Universal Robots PolyScope program: 0622_1902.urp

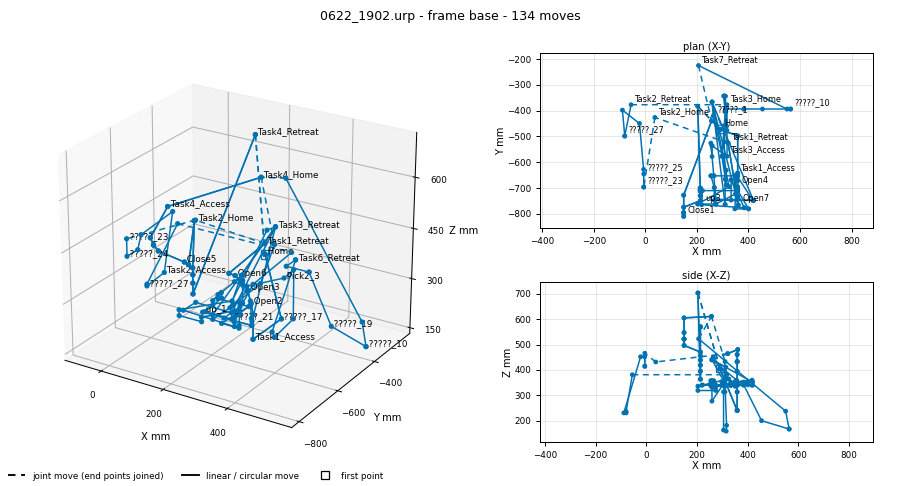
[picture p0: tool path of 0622_1902.urp in frame base, 134 of 134 moves have a stored position in this frame; points joined in program order, loops and branches not executed]
Program 0622_1902 (installation=default directory=/programs/usbdisk/새로운 폴더_3 createdIn=5.12.7.1102192 lastSavedIn=5.11.0.108249 robotSerialNumber=20215501208)
Calibrated DH parameters: a=[0.000135, -0.201821, -0.391913, -0.000063, 0.000038, 0]; d=[0.162484, -479.507804, 481.562221, -1.92078, 0.099549, 0.099572]; alpha=[1.570789, -0.00078, 0.007148, 1.569147, -1.569841, 0]; deltaTheta=[0, 1.075971, -1.038513, -0.037456, 0, 0]
Robot Program (runOnlyOnce=false)
  Folder Init
    Call Init_Variables
    Script: global repeat = 0
    Call Socket_Open
    MoveJ speed 60 deg/s, acceleration 80 deg/s^2 (useActiveTCP=true) feature=Base
      Waypoint Home: TCP in base x=290.307 y=-472.673 z=405.346 mm, rx=-2.2604 ry=-2.147 rz=0.0783 rad; joints [-251.839, -82.418, 93.917, 258.527, -92.811, 111.318] deg
    Wait Sleep waitTime=1
  Loop Forever
    Folder Main Sequence
      Folder Task1:OpenPrinter
        Call Enter_Next_Task
        Loop While (checkContinuously=false) expression=retry_count <= max_retry and task_done == 0
          MoveJ speed 60 deg/s, acceleration 80 deg/s^2 (useActiveTCP=true) feature=Base
            Waypoint Task1_Home: TCP in base x=290.314 y=-472.7 z=405.337 mm, rx=-2.2604 ry=-2.147 rz=0.0783 rad; joints [-251.84, -82.414, 93.913, 258.528, -92.81, 111.316] deg
          MoveL speed 250 mm/s, acceleration 1200 mm/s^2 (useActiveTCP=true) feature=Base
            Waypoint 웨이포인트_17: TCP in base x=358.108 y=-497.437 z=239.959 mm, rx=-2.2605 ry=-2.1469 rz=0.0783 rad; joints [-246.378, -66.361, 98.95, 237.748, -92.865, 116.914] deg
            Waypoint Task1_Access: TCP in base x=358.145 y=-643.31 z=239.914 mm, rx=-2.2603 ry=-2.1469 rz=0.0783 rad; joints [-250.947, -51.356, 74.514, 246.926, -92.843, 112.267] deg
          MoveL speed 250 mm/s, acceleration 1200 mm/s^2 (useActiveTCP=true) feature=Base
            Waypoint Open1: TCP in base x=358.112 y=-643.249 z=312.941 mm, rx=-2.2756 ry=-2.1607 rz=0.0433 rad; joints [-251.165, -54.868, 69.274, 255.167, -91.168, 112.004] deg
            Waypoint Open2: TCP in base x=358.116 y=-653.358 z=348.764 mm, rx=-2.2399 ry=-2.1285 rz=-0.0282 rad; joints [-251.571, -53.878, 61.395, 265.654, -89.944, 111.495] deg
            Waypoint Open3: TCP in base x=358.131 y=-671.047 z=394.191 mm, rx=-2.2065 ry=-2.0982 rz=-0.0914 rad; joints [-252.118, -50.739, 48.753, 278.451, -88.91, 110.769] deg
            Waypoint Open4: TCP in base x=358.139 y=-695.842 z=432.417 mm, rx=-2.2066 ry=-2.0983 rz=-0.0912 rad; joints [-252.66, -45.306, 33.722, 288.051, -88.986, 110.159] deg
            Waypoint Open5: TCP in base x=358.138 y=-703.871 z=432.339 mm, rx=2.1752 ry=2.0611 rz=-0.2397 rad; joints [-252.159, -50.267, 46.998, 262.355, -94.486, 110.613] deg
            Waypoint Open6: TCP in base x=358.152 y=-732.149 z=460.497 mm, rx=2.1751 ry=2.0611 rz=-0.2398 rad; joints [-252.775, -44.157, 32.21, 270.972, -94.36, 109.938] deg
            Waypoint Open7: TCP in base x=360.469 y=-765.799 z=480.398 mm, rx=2.1073 ry=1.9941 rz=-0.3503 rad; joints [-253.083, -35.969, 16.049, 272.511, -96.174, 109.139] deg
          MoveL speed 250 mm/s, acceleration 1200 mm/s^2 (useActiveTCP=true) feature=Base
            Waypoint Task1_Retreat: TCP in base x=320.913 y=-525.366 z=464.12 mm, rx=-2.2348 ry=-2.2055 rz=-0.1004 rad; joints [-251.676, -74.86, 75.667, 270.873, -86.355, 109.144] deg
          Wait Sleep waitTime=1
          SuppressedNode
            Call Check_Door_Open
          SuppressedNode
            Switch expression=fail_flag
              Case (caseValue=0)
                Script: task_done = 1
              Case (caseValue=1)
                Script: retry_count = retry_count + 1
          Call Check_Camera_Open
          Switch expression=fail_flag
            Case (caseValue=0)
              Script: task_done = 1
            Case (caseValue=1)
              Script: retry_count = retry_count + 1
        If task_done == 0
          Call Error_Stop
        Wait Sleep waitTime=1
      Folder Task2,3,3+:PickAndPlace
        Call Enter_Next_Task
        Loop While (checkContinuously=false) expression=nopaper == 1
          Loop While (checkContinuously=false) expression=retry_count <= max_retry and task_done == 0
            Folder Task2:PickA4FromTray
              MoveJ speed 60 deg/s, acceleration 80 deg/s^2 (useActiveTCP=true) feature=Base
                Waypoint Task2_Home: TCP in base x=36.96 y=-426.094 z=431.249 mm, rx=1.9338 ry=1.8099 rz=-0.6845 rad; joints [-284.402, -104.722, 122.782, 215.162, -85.651, 81.217] deg
              Call Gripper_Open
              Call Wait_Motor_Idle
              Folder 폴더
                MoveJ speed 60 deg/s, acceleration 80 deg/s^2 (useActiveTCP=true) feature=Base
                  Waypoint 웨이포인트_23: TCP in base x=-6.335 y=-696.326 z=465.636 mm, rx=2.2415 ry=-0.3574 rz=-0.16 rad; joints [-280.885, -66.992, 81.728, 205.322, -95.11, 185.235] deg
                MoveL speed 250 mm/s, acceleration 1200 mm/s^2 (useActiveTCP=true) feature=Base
                  Waypoint 웨이포인트_24: TCP in base x=-6.322 y=-696.307 z=414.387 mm, rx=2.2415 ry=-0.3575 rz=-0.16 rad; joints [-280.889, -64.814, 86.427, 198.445, -95.156, 185.249] deg
                  Waypoint 웨이포인트_25: TCP in base x=-6.303 y=-645.419 z=414.389 mm, rx=2.2414 ry=-0.3575 rz=-0.16 rad; joints [-281.881, -71.275, 95.746, 195.526, -94.416, 184.618] deg
                  Waypoint 웨이포인트_28: TCP in base x=-6.918 y=-627.811 z=451.854 mm, rx=2.2414 ry=-0.3575 rz=-0.1599 rad; joints [-282.329, -75.473, 95.437, 200.006, -94.042, 184.326] deg
              MoveL speed 250 mm/s, acceleration 1200 mm/s^2 (useActiveTCP=true) feature=Base
                Waypoint 웨이포인트_26: TCP in base x=-22.834 y=-449.606 z=451.838 mm, rx=2.2414 ry=-0.3575 rz=-0.1599 rad; joints [-290.868, -100.504, 121.499, 198.842, -87.496, 178.874] deg
                Waypoint Task2_Access: TCP in base x=-89.035 y=-397.687 z=230.223 mm, rx=1.5681 ry=0.0538 rz=0.0669 rad; joints [-313.235, -57.01, 139.142, 97.671, -42.763, 180.679] deg
                Waypoint 웨이포인트_27: TCP in base x=-80.06 y=-498.27 z=230.219 mm, rx=1.5682 ry=0.0538 rz=0.067 rad; joints [-301.557, -52.728, 123.378, 109.146, -54.422, 180.732] deg
                Waypoint 웨이포인트_12: TCP in base x=-80.054 y=-498.26 z=235.695 mm, rx=1.5681 ry=0.0538 rz=0.0669 rad; joints [-301.558, -53.562, 123.445, 109.909, -54.42, 180.737] deg
              Wait Sleep waitTime=1
              Call Gripper_Close
              Call Wait_Motor_Idle
              MoveL speed 250 mm/s, acceleration 1200 mm/s^2 (useActiveTCP=true) feature=Base
                Waypoint Task2_Retreat: TCP in base x=-55.478 y=-376.727 z=380.943 mm, rx=1.5681 ry=0.0539 rz=0.0669 rad; joints [-310.988, -89.069, 140.295, 128.379, -44.954, 180.96] deg
              If fail_flag == 1
                Call Error_Stop
              Wait Sleep waitTime=3
            Folder Task3:PlaceA4OnScanner
              Call Enter_Next_Task
              MoveJ speed 60 deg/s, acceleration 80 deg/s^2 (useActiveTCP=true) feature=Base
                Waypoint Task3_Home: TCP in base x=316.751 y=-376.736 z=380.91 mm, rx=1.5682 ry=0.054 rz=0.0668 rad; joints [-240.78, -72.729, 119.686, 133.121, -115.13, 180.786] deg
              MoveL speed 250 mm/s, acceleration 1200 mm/s^2 (useActiveTCP=true) feature=Base
                Waypoint Task3_Access: TCP in base x=316.801 y=-576.799 z=363.883 mm, rx=1.5682 ry=0.054 rz=0.067 rad; joints [-250.736, -54.554, 93.02, 141.565, -105.113, 180.827] deg
              MoveL speed 250 mm/s, acceleration 1200 mm/s^2 (useActiveTCP=true) feature=Base
                Waypoint Place1: TCP in base x=258.695 y=-535.855 z=276.647 mm, rx=1.5682 ry=0.0539 rz=0.067 rad; joints [-255.555, -52.152, 107.026, 125.111, -100.371, 180.737] deg
                Waypoint Place2: TCP in base x=258.714 y=-535.837 z=330.851 mm, rx=1.9481 ry=0.0428 rz=0.0806 rad; joints [-255.789, -65.713, 110.061, 157.638, -98.984, 186.181] deg
                Waypoint Place3: TCP in base x=258.706 y=-577.686 z=357.608 mm, rx=2.0696 ry=0.0386 rz=0.0849 rad; joints [-257.026, -66.21, 102.611, 172.482, -97.075, 187.174] deg
              Call Gripper_Open
              Call Wait_Motor_Idle
              MoveL speed 250 mm/s, acceleration 1200 mm/s^2 (useActiveTCP=true) feature=Base
                Waypoint 웨이포인트_6: TCP in base x=254.047 y=-525.754 z=357.577 mm, rx=2.1241 ry=0.0396 rz=0.0817 rad; joints [-256.235, -72.651, 110.764, 173.964, -97.528, 187.976] deg
                Waypoint 웨이포인트_7: TCP in base x=265.506 y=-653.622 z=357.598 mm, rx=2.124 ry=0.0397 rz=0.0817 rad; joints [-258.032, -58.705, 89.296, 181.36, -95.938, 187.013] deg
                Waypoint 웨이포인트_8: TCP in base x=265.302 y=-651.492 z=340.681 mm, rx=2.124 ry=0.0397 rz=0.0817 rad; joints [-258.01, -57.739, 90.591, 179.098, -95.971, 187.023] deg
                Waypoint 웨이포인트_13: TCP in base x=273.53 y=-743.632 z=340.722 mm, rx=2.124 ry=0.0397 rz=0.0817 rad; joints [-258.911, -46.995, 71.73, 187.158, -95.142, 186.541] deg
                Waypoint 웨이포인트_21: TCP in base x=356.126 y=-746.074 z=340.698 mm, rx=2.124 ry=0.0397 rz=0.0818 rad; joints [-252.554, -42.043, 62.558, 191.888, -100.492, 189.948] deg
                Waypoint 웨이포인트_29: TCP in base x=356.13 y=-746.059 z=359.504 mm, rx=2.124 ry=0.0397 rz=0.0817 rad; joints [-252.552, -43.007, 61.421, 193.988, -100.482, 189.944] deg
              MoveL speed 250 mm/s, acceleration 1200 mm/s^2 (useActiveTCP=true) feature=Base
                Waypoint Task3_Retreat: TCP in base x=258.692 y=-366.204 z=439.923 mm, rx=2.1237 ry=0.0367 rz=0.0867 rad; joints [-249.2, -96.96, 123.493, 186.236, -103.267, 192.051] deg
              Wait Sleep waitTime=1
              Call Check_Camera_Align
              Switch expression=paper_state
                Case (caseValue=0)
                  Script: retry_count = retry_count + 1
                Case (caseValue=1)
                  Script: task_done = 1
              Wait Sleep waitTime=1
          If task_done == 0
            Call Error_Stop
          Folder Task3+:PaperAlign
            Wait Sleep waitTime=1
            Call Check_Camera_Align
            Loop While (checkContinuously=false) expression=paper_align_state != 0 and paper_align_state != 9 and align_retry_count <= max_retry
              Script: align_retry_count = align_retry_count + 1
              MoveL speed 250 mm/s, acceleration 1200 mm/s^2 (useActiveTCP=true) feature=Base
                Waypoint 웨이포인트_1: TCP in base x=263.645 y=-419.544 z=450.752 mm, rx=2.1095 ry=0.0567 rz=0.0671 rad; joints [-251.124, -90.818, 116.42, 186.206, -102.101, 189.536] deg
                Waypoint 웨이포인트_5: TCP in base x=325.163 y=-694.866 z=364.547 mm, rx=2.1237 ry=0.0368 rz=0.0868 rad; joints [-253.782, -51.437, 75.758, 187.916, -99.351, 189.514] deg
              Switch expression=paper_align_state
                Case (caseValue=1)
                  SuppressedNode
                    MoveL speed 250 mm/s, acceleration 1200 mm/s^2 (useActiveTCP=true) feature=Base
                      Waypoint home_up: TCP in base x=411.069 y=-776.712 z=349.862 mm, rx=2.1238 ry=0.0368 rz=0.0867 rad; joints [-249.41, -33.925, 45.774, 200.882, -102.945, 191.884] deg
                      Waypoint touch: TCP in base x=411.033 y=-776.714 z=334.504 mm, rx=2.1236 ry=0.0367 rz=0.0867 rad; joints [-249.413, -33.291, 46.859, 199.158, -102.957, 191.886] deg
                      Waypoint down: TCP in base x=313.835 y=-617.619 z=339.178 mm, rx=2.1238 ry=0.0367 rz=0.0868 rad; joints [-252.767, -58.652, 92.334, 178.663, -100.285, 190.075] deg
                      Waypoint right: TCP in base x=250.722 y=-620.02 z=338.484 mm, rx=2.1239 ry=0.0366 rz=0.0869 rad; joints [-258.809, -61.528, 97.303, 176.099, -95.176, 186.838] deg
                      Waypoint up: TCP in base x=245.21 y=-744.892 z=339.67 mm, rx=2.1238 ry=0.0367 rz=0.0868 rad; joints [-261.255, -48.066, 73.863, 185.967, -93.018, 185.539] deg
                      Waypoint left: TCP in base x=408.353 y=-753.62 z=337.643 mm, rx=2.1235 ry=0.0364 rz=0.0868 rad; joints [-248.997, -37.091, 53.665, 196.203, -103.338, 192.136] deg
                      Waypoint z_up: TCP in base x=408.373 y=-753.612 z=350.303 mm, rx=2.1236 ry=0.0365 rz=0.0868 rad; joints [-248.995, -37.678, 52.851, 197.607, -103.325, 192.135] deg
                  SuppressedNode
                    MoveL speed 250 mm/s, acceleration 1200 mm/s^2 (useActiveTCP=true) feature=Base
                      Waypoint top_home: TCP in base x=476.403 y=-777.08 z=332.173 mm, rx=2.0259 ry=0.0603 rz=0.0427 rad; joints [-244.874, -24.378, 31.553, 200.812, -109.067, 190.542] deg
                      Waypoint lefttop1: TCP in base x=476.428 y=-777.056 z=326.289 mm, rx=2.0258 ry=0.0603 rz=0.0427 rad; joints [-244.872, -24.18, 32.025, 200.14, -109.072, 190.543] deg
                      Waypoint lefttop2: TCP in base x=418.211 y=-735.241 z=318.888 mm, rx=2.0259 ry=0.0603 rz=0.0427 rad; joints [-247.527, -36.33, 57.095, 186.808, -106.819, 189.265] deg
                      Waypoint lefttop3: TCP in base x=418.224 y=-735.252 z=329.315 mm, rx=2.0259 ry=0.0603 rz=0.0428 rad; joints [-247.527, -36.912, 56.59, 187.895, -106.81, 189.264] deg
                      Waypoint lefttop4: TCP in base x=476.403 y=-777.08 z=332.173 mm, rx=2.0259 ry=0.0603 rz=0.0427 rad; joints [-244.874, -24.378, 31.553, 200.812, -109.067, 190.542] deg
                      Waypoint lefttop5: TCP in base x=476.428 y=-777.056 z=326.289 mm, rx=2.0258 ry=0.0603 rz=0.0427 rad; joints [-244.872, -24.18, 32.025, 200.14, -109.072, 190.543] deg
                      Waypoint lefttop6: TCP in base x=418.249 y=-735.21 z=317.328 mm, rx=2.0257 ry=0.0603 rz=0.0428 rad; joints [-247.524, -36.239, 57.167, 186.634, -106.822, 189.262] deg
                      Waypoint 웨이포인트_34: TCP in base x=254.455 y=-652.624 z=348.54 mm, rx=2.1239 ry=0.0371 rz=0.0867 rad; joints [-259.06, -58.691, 90.844, 179.708, -94.929, 186.683] deg
                      Waypoint move_to_right: TCP in base x=316.854 y=-733.109 z=330.021 mm, rx=2.0257 ry=-0.0559 rz=-0.0297 rad; joints [-254.229, -43.603, 69.178, 181.965, -106.74, 189.197] deg
                      Waypoint righttop_home: TCP in base x=198.901 y=-787.594 z=329.962 mm, rx=2.018 ry=-0.2066 rz=-0.1238 rad; joints [-263.364, -41.811, 65.831, 183.44, -106.194, 188.908] deg
                      Waypoint righttop1: TCP in base x=198.92 y=-787.585 z=321.803 mm, rx=2.018 ry=-0.2066 rz=-0.1238 rad; joints [-263.362, -41.311, 66.196, 182.574, -106.201, 188.907] deg
                      Waypoint righttop2: TCP in base x=198.916 y=-755.326 z=321.817 mm, rx=2.0181 ry=-0.2066 rz=-0.1237 rad; joints [-263.056, -45.33, 73.758, 179.077, -106.5, 189.056] deg
                      Waypoint 웨이포인트_35: TCP in base x=267.387 y=-698.175 z=352.437 mm, rx=2.1237 ry=0.0371 rz=0.0866 rad; joints [-258.698, -53.341, 81.09, 184.124, -95.208, 186.872] deg
                      Waypoint righttop_home: TCP in base x=198.901 y=-787.594 z=329.962 mm, rx=2.018 ry=-0.2066 rz=-0.1238 rad; joints [-263.364, -41.811, 65.831, 183.44, -106.194, 188.908] deg
                      Waypoint righttop1: TCP in base x=198.92 y=-787.585 z=321.803 mm, rx=2.018 ry=-0.2066 rz=-0.1238 rad; joints [-263.362, -41.311, 66.196, 182.574, -106.201, 188.907] deg
                      Waypoint righttop2: TCP in base x=198.916 y=-755.326 z=321.817 mm, rx=2.0181 ry=-0.2066 rz=-0.1237 rad; joints [-263.056, -45.33, 73.758, 179.077, -106.5, 189.056] deg
                      Waypoint 웨이포인트_35: TCP in base x=267.387 y=-698.175 z=352.437 mm, rx=2.1237 ry=0.0371 rz=0.0866 rad; joints [-258.698, -53.341, 81.09, 184.124, -95.208, 186.872] deg
                      Waypoint 웨이포인트_36: TCP in base x=267.318 y=-698.171 z=339.177 mm, rx=2.1237 ry=0.0369 rz=0.0866 rad; joints [-258.704, -52.477, 81.792, 182.558, -95.216, 186.875] deg
                      Waypoint 웨이포인트_37: TCP in base x=378.814 y=-710.052 z=321.31 mm, rx=2.0182 ry=-0.2066 rz=-0.1238 rad; joints [-247.983, -41.401, 65.997, 186.167, -119.675, 197.015] deg
                      Waypoint 웨이포인트_38: TCP in base x=378.85 y=-764.571 z=321.307 mm, rx=2.0182 ry=-0.2066 rz=-0.1238 rad; joints [-249.486, -34.393, 52.607, 192.111, -118.328, 196.135] deg
                      Waypoint 웨이포인트_39: TCP in base x=378.79 y=-764.605 z=321.308 mm, rx=2.0182 ry=-0.2067 rz=-0.1239 rad; joints [-249.491, -34.393, 52.605, 192.113, -118.329, 196.133] deg
                  MoveL speed 250 mm/s, acceleration 1200 mm/s^2 (useActiveTCP=true) feature=Base
                    Waypoint out_top_home_1: TCP in base x=203.102 y=-761.983 z=335.486 mm, rx=2.0028 ry=-0.2108 rz=-0.1158 rad; joints [-262.793, -45.047, 71.304, 180.396, -106.628, 189.392] deg
                    Waypoint out_top_touch_1: TCP in base x=203.111 y=-761.964 z=318.614 mm, rx=2.0027 ry=-0.2108 rz=-0.1159 rad; joints [-262.792, -43.949, 72.027, 178.57, -106.643, 189.389] deg
                    Waypoint out_top_left_1: TCP in base x=273.333 y=-761.997 z=318.66 mm, rx=2.0026 ry=-0.2109 rz=-0.1159 rad; joints [-257.196, -40.917, 66.151, 182.335, -111.608, 192.092] deg
                    Waypoint out_top_z_up_1: TCP in base x=273.301 y=-762.006 z=331.73 mm, rx=2.0027 ry=-0.2109 rz=-0.1159 rad; joints [-257.198, -41.724, 65.578, 183.721, -111.597, 192.093] deg
                    Waypoint out_top_home_2: TCP in base x=350.147 y=-722.859 z=353.835 mm, rx=2.1236 ry=0.0368 rz=0.0867 rad; joints [-252.473, -46.032, 67.835, 190.561, -100.442, 190.217] deg
                    Waypoint out_top_touch_2: TCP in base x=350.162 y=-722.849 z=335.209 mm, rx=2.1236 ry=0.0368 rz=0.0868 rad; joints [-252.473, -44.979, 68.869, 188.473, -100.452, 190.221] deg
                    Waypoint down_1: TCP in base x=350.105 y=-652.862 z=337.787 mm, rx=2.1238 ry=0.0368 rz=0.0868 rad; joints [-250.62, -52.889, 82.637, 182.839, -102.064, 191.242] deg
                    Waypoint right_1: TCP in base x=254.42 y=-652.638 z=336.904 mm, rx=2.1238 ry=0.037 rz=0.0867 rad; joints [-259.063, -57.835, 91.436, 178.254, -94.94, 186.683] deg
                    Waypoint 웨이포인트_34: TCP in base x=254.455 y=-652.624 z=348.54 mm, rx=2.1239 ry=0.0371 rz=0.0867 rad; joints [-259.06, -58.691, 90.844, 179.708, -94.929, 186.683] deg
                    Waypoint 웨이포인트_35: TCP in base x=267.387 y=-698.175 z=352.437 mm, rx=2.1237 ry=0.0371 rz=0.0866 rad; joints [-258.698, -53.341, 81.09, 184.124, -95.208, 186.872] deg
                    Waypoint 웨이포인트_36: TCP in base x=267.318 y=-698.171 z=339.177 mm, rx=2.1237 ry=0.0369 rz=0.0866 rad; joints [-258.704, -52.477, 81.792, 182.558, -95.216, 186.875] deg
                    Waypoint up_1: TCP in base x=267.384 y=-747.516 z=339.193 mm, rx=2.1237 ry=0.037 rz=0.0867 rad; joints [-259.485, -46.723, 71.497, 187.057, -94.512, 186.455] deg
                    Waypoint left_1: TCP in base x=417.039 y=-747.555 z=339.153 mm, rx=2.1238 ry=0.0369 rz=0.0866 rad; joints [-248.23, -37.306, 53.822, 196.381, -103.973, 192.544] deg
                    Waypoint z_up_2: TCP in base x=417.042 y=-747.569 z=359.498 mm, rx=2.1237 ry=0.0369 rz=0.0866 rad; joints [-248.228, -38.218, 52.46, 198.653, -103.963, 192.541] deg
                Case (caseValue=2)
                  MoveL speed 250 mm/s, acceleration 1200 mm/s^2 (useActiveTCP=true) feature=Base
                    Waypoint out_down_home: motionParameters(nextMotionTime=2); TCP in base x=353.061 y=-649.128 z=353.349 mm, rx=2.1237 ry=0.0367 rz=0.0867 rad; joints [-250.263, -54.126, 82.18, 184.573, -102.361, 191.44] deg
                    Waypoint out_down_touch: TCP in base x=353.03 y=-649.115 z=339.829 mm, rx=2.1237 ry=0.0367 rz=0.0867 rad; joints [-250.265, -53.239, 82.9, 182.965, -102.368, 191.441] deg
                    Waypoint up2: TCP in base x=347.298 y=-780.895 z=340.744 mm, rx=2.1237 ry=0.0368 rz=0.0868 rad; joints [-253.981, -37.91, 54.824, 195.3, -99.119, 189.395] deg
                    Waypoint left2: TCP in base x=400.466 y=-780.911 z=340.74 mm, rx=2.1237 ry=0.0368 rz=0.0868 rad; joints [-250.239, -33.821, 46.958, 199.482, -102.253, 191.428] deg
                    Waypoint z_up2: TCP in base x=400.454 y=-780.931 z=348.394 mm, rx=2.1237 ry=0.0369 rz=0.0868 rad; joints [-250.24, -34.134, 46.411, 200.345, -102.244, 191.425] deg
                Case (caseValue=3)
                  MoveL speed 250 mm/s, acceleration 1200 mm/s^2 (useActiveTCP=true) feature=Base
                    Waypoint out_left_home: TCP in base x=358.429 y=-710.028 z=350.153 mm, rx=2.1239 ry=0.0369 rz=0.0868 rad; joints [-251.517, -46.844, 69.865, 189.462, -101.252, 190.743] deg
                    Waypoint out_left_touch: TCP in base x=358.445 y=-710.017 z=338.142 mm, rx=2.1238 ry=0.0369 rz=0.0868 rad; joints [-251.516, -46.149, 70.523, 188.107, -101.261, 190.744] deg
                    Waypoint right3: TCP in base x=221.511 y=-710.02 z=340.705 mm, rx=2.1237 ry=0.0369 rz=0.0868 rad; joints [-262.859, -53.18, 82.791, 182.099, -91.678, 184.689] deg
                    Waypoint up3: TCP in base x=218.375 y=-764.918 z=339.146 mm, rx=2.1237 ry=0.037 rz=0.0871 rad; joints [-263.669, -46.658, 71.407, 186.948, -90.935, 184.26] deg
                    Waypoint left3: TCP in base x=383.557 y=-776.618 z=339.385 mm, rx=2.1238 ry=0.0368 rz=0.0868 rad; joints [-251.307, -35.82, 51.011, 197.308, -101.368, 190.849] deg
                    Waypoint z_up3: TCP in base x=383.557 y=-776.624 z=352.28 mm, rx=2.1238 ry=0.0368 rz=0.0868 rad; joints [-251.306, -36.385, 50.141, 198.744, -101.361, 190.845] deg
                Case (caseValue=4)
                  MoveL speed 250 mm/s, acceleration 1200 mm/s^2 (useActiveTCP=true) feature=Base
                    Waypoint out_right_home: TCP in base x=332.757 y=-668.076 z=351.636 mm, rx=2.1238 ry=0.0368 rz=0.0868 rad; joints [-252.488, -53.205, 80.911, 184.667, -100.474, 190.221] deg
                    Waypoint out_right_touch: TCP in base x=332.745 y=-668.072 z=339.134 mm, rx=2.1237 ry=0.0367 rz=0.0868 rad; joints [-252.489, -52.39, 81.569, 183.19, -100.483, 190.22] deg
                    Waypoint up4: TCP in base x=332.784 y=-746.83 z=338.35 mm, rx=2.1237 ry=0.0369 rz=0.0869 rad; joints [-254.346, -43.281, 65.261, 190.205, -98.848, 189.205] deg
                    Waypoint left4: TCP in base x=419.342 y=-748.177 z=339.772 mm, rx=2.1238 ry=0.037 rz=0.0869 rad; joints [-248.089, -37.058, 53.254, 196.721, -104.078, 192.627] deg
                    Waypoint z_up4: TCP in base x=419.35 y=-748.182 z=351.876 mm, rx=2.1238 ry=0.037 rz=0.0869 rad; joints [-248.088, -37.609, 52.459, 198.068, -104.069, 192.625] deg
              MoveL speed 250 mm/s, acceleration 1200 mm/s^2 (useActiveTCP=true) feature=Base
                Waypoint Task3_Retreat: TCP in base x=258.692 y=-366.204 z=439.923 mm, rx=2.1237 ry=0.0367 rz=0.0867 rad; joints [-249.2, -96.96, 123.493, 186.236, -103.267, 192.051] deg
              Wait Sleep waitTime=1
              Call Check_Camera_Align
            If paper_align_state != 0
              Loop Counting (count=3) loopVariable(name=루프_11)
                MoveL speed 250 mm/s, acceleration 1200 mm/s^2 (useActiveTCP=true) feature=Base
                  Waypoint clr_scanner_1: TCP in base x=309.352 y=-764.14 z=348.523 mm, rx=2.1236 ry=0.0365 rz=0.0869 rad; joints [-256.47, -42.967, 63.114, 191.858, -97.043, 188.077] deg
                  Waypoint clr_scanner_2: TCP in base x=309.355 y=-764.127 z=335.554 mm, rx=2.1235 ry=0.0365 rz=0.0868 rad; joints [-256.47, -42.268, 63.85, 190.42, -97.054, 188.076] deg
                  Waypoint clr_scanner_3: TCP in base x=309.342 y=-666.018 z=335.451 mm, rx=2.1237 ry=0.0365 rz=0.0868 rad; joints [-254.423, -53.641, 84.415, 181.402, -98.862, 189.183] deg
                  Waypoint clr_scanner_4: TCP in base x=305.938 y=-521.343 z=341.67 mm, rx=2.1236 ry=0.0365 rz=0.0868 rad; joints [-250.41, -68.645, 107.812, 173.436, -102.327, 191.373] deg
                  Waypoint clr_scanner_5: TCP in base x=310.318 y=-457.04 z=432.696 mm, rx=2.1236 ry=0.0365 rz=0.0868 rad; joints [-247.191, -81.97, 109.48, 185.54, -104.959, 193.179] deg
              Script: global nopaper = 1
              Script: global task_done = 0
            Else 
              Script: global nopaper = 0
            If paper_align_state == 0
              Script: nopaper = 0
      Folder Task4:ClosePrinter
        Call Enter_Next_Task
        Loop While (checkContinuously=false) expression=retry_count <= max_retry and task_done == 0
          MoveJ speed 60 deg/s, acceleration 80 deg/s^2 (useActiveTCP=true) feature=Base
            Waypoint Task4_Home: TCP in base x=256.826 y=-439.474 z=610.895 mm, rx=2.3079 ry=0.0086 rz=0.0018 rad; joints [-252.464, -94.611, 91.606, 226.691, -102.422, 192.055] deg
          MoveL speed 250 mm/s, acceleration 1200 mm/s^2 (useActiveTCP=true) feature=Base
            Waypoint Task4_Access: TCP in base x=148.636 y=-727.715 z=605.166 mm, rx=1.2884 ry=-1.2507 rz=1.1591 rad; joints [-268.772, -57.066, 57.637, 184.345, -90.714, 269.314] deg
          MoveL speed 250 mm/s, acceleration 1200 mm/s^2 (useActiveTCP=true) feature=Base
            Waypoint Close1: TCP in base x=148.688 y=-809.891 z=547.115 mm, rx=1.4249 ry=-1.385 rz=1.0616 rad; joints [-268.907, -45.466, 43.512, 197.581, -90.443, 269.491] deg
            Waypoint Close2: TCP in base x=148.64 y=-796.037 z=521.65 mm, rx=1.4248 ry=-1.385 rz=1.0616 rad; joints [-268.893, -47.909, 51.494, 192.04, -90.504, 269.502] deg
            Waypoint Close3: TCP in base x=148.649 y=-796.055 z=521.571 mm, rx=1.6083 ry=-1.5658 rz=0.9063 rad; joints [-268.903, -50.476, 50.97, 209.943, -90.274, 269.718] deg
            Waypoint Close4: TCP in base x=148.687 y=-774.487 z=496.375 mm, rx=1.6083 ry=-1.5657 rz=0.9065 rad; joints [-268.873, -53.722, 60.073, 204.08, -90.336, 269.753] deg
            Waypoint Close5: TCP in base x=213.156 y=-749.245 z=470.417 mm, rx=1.6082 ry=-1.5657 rz=0.9065 rad; joints [-263.371, -54.366, 64.948, 200.023, -95.109, 272.561] deg
            Waypoint Close6: TCP in base x=213.168 y=-729.713 z=455.466 mm, rx=1.5446 ry=-1.5029 rz=0.9638 rad; joints [-263.137, -55.596, 71.043, 189.957, -95.666, 272.141] deg
            Waypoint 웨이포인트_2: TCP in base x=213.168 y=-700.447 z=569.635 mm, rx=1.5446 ry=-1.5029 rz=0.9637 rad; joints [-262.813, -62.268, 64.571, 203.117, -95.876, 272.261] deg
            Waypoint 웨이포인트_3: TCP in base x=213.139 y=-700.438 z=569.664 mm, rx=0.7687 ry=-0.7398 rz=1.4198 rad; joints [-262.888, -44.099, 47.902, 141.673, -95.592, 265.105] deg
            Waypoint 웨이포인트_4: TCP in base x=213.129 y=-710.201 z=438.633 mm, rx=0.7687 ry=-0.7398 rz=1.4198 rad; joints [-262.988, -38.166, 56.593, 127.044, -95.578, 265.084] deg
            Waypoint 웨이포인트_14: TCP in base x=213.137 y=-710.216 z=418.872 mm, rx=0.9791 ry=-0.9464 rz=1.3335 rad; joints [-262.867, -42.891, 66.704, 137.401, -96.512, 266.805] deg
            Waypoint 웨이포인트_15: TCP in base x=213.142 y=-710.217 z=394.52 mm, rx=1.1095 ry=-1.0745 rz=1.2674 rad; joints [-262.827, -44.827, 72.245, 143.715, -96.823, 268.018] deg
            Waypoint 웨이포인트_16: TCP in base x=213.146 y=-710.207 z=363.102 mm, rx=1.1858 ry=-1.1496 rz=1.2239 rad; joints [-262.817, -44.652, 75.673, 145.981, -96.899, 268.757] deg
          MoveL speed 250 mm/s, acceleration 1200 mm/s^2 (useActiveTCP=true) feature=Base
            Waypoint Task4_Retreat: TCP in base x=203.304 y=-382.609 z=703.619 mm, rx=0.9532 ry=-1.0966 rz=1.2827 rad; joints [-255.678, -95.084, 95.274, 165.571, -108.944, 268.685] deg
          Wait Sleep waitTime=1
          Call Check_Door_Closed
          Switch expression=fail_flag
            Case (caseValue=0)
              Script: task_done = 1
            Case (caseValue=1)
              Script: retry_count = retry_count + 1
        If task_done == 0
          Call Error_Stop
        Wait Sleep waitTime=1
      Folder Task1:OpenPrinter
        Call Enter_Next_Task
        Loop While (checkContinuously=false) expression=retry_count <= max_retry and task_done == 0
          MoveJ speed 60 deg/s, acceleration 80 deg/s^2 (useActiveTCP=true) feature=Base
            Waypoint Task1_Home: TCP in base x=290.314 y=-472.7 z=405.337 mm, rx=-2.2604 ry=-2.147 rz=0.0783 rad; joints [-251.84, -82.414, 93.913, 258.528, -92.81, 111.316] deg
          MoveL speed 250 mm/s, acceleration 1200 mm/s^2 (useActiveTCP=true) feature=Base
            Waypoint 웨이포인트_17: TCP in base x=358.108 y=-497.437 z=239.959 mm, rx=-2.2605 ry=-2.1469 rz=0.0783 rad; joints [-246.378, -66.361, 98.95, 237.748, -92.865, 116.914] deg
            Waypoint Task1_Access: TCP in base x=358.145 y=-643.31 z=239.914 mm, rx=-2.2603 ry=-2.1469 rz=0.0783 rad; joints [-250.947, -51.356, 74.514, 246.926, -92.843, 112.267] deg
          MoveL speed 250 mm/s, acceleration 1200 mm/s^2 (useActiveTCP=true) feature=Base
            Waypoint Open1: TCP in base x=358.112 y=-643.249 z=312.941 mm, rx=-2.2756 ry=-2.1607 rz=0.0433 rad; joints [-251.165, -54.868, 69.274, 255.167, -91.168, 112.004] deg
            Waypoint Open2: TCP in base x=358.116 y=-653.358 z=348.764 mm, rx=-2.2399 ry=-2.1285 rz=-0.0282 rad; joints [-251.571, -53.878, 61.395, 265.654, -89.944, 111.495] deg
            Waypoint Open3: TCP in base x=358.131 y=-671.047 z=394.191 mm, rx=-2.2065 ry=-2.0982 rz=-0.0914 rad; joints [-252.118, -50.739, 48.753, 278.451, -88.91, 110.769] deg
            Waypoint Open4: TCP in base x=358.139 y=-695.842 z=432.417 mm, rx=-2.2066 ry=-2.0983 rz=-0.0912 rad; joints [-252.66, -45.306, 33.722, 288.051, -88.986, 110.159] deg
            Waypoint Open5: TCP in base x=358.138 y=-703.871 z=432.339 mm, rx=2.1752 ry=2.0611 rz=-0.2397 rad; joints [-252.159, -50.267, 46.998, 262.355, -94.486, 110.613] deg
            Waypoint Open6: TCP in base x=358.152 y=-732.149 z=460.497 mm, rx=2.1751 ry=2.0611 rz=-0.2398 rad; joints [-252.775, -44.157, 32.21, 270.972, -94.36, 109.938] deg
            Waypoint Open7: TCP in base x=360.469 y=-765.799 z=480.398 mm, rx=2.1073 ry=1.9941 rz=-0.3503 rad; joints [-253.083, -35.969, 16.049, 272.511, -96.174, 109.139] deg
          MoveL speed 250 mm/s, acceleration 1200 mm/s^2 (useActiveTCP=true) feature=Base
            Waypoint Task1_Retreat: TCP in base x=320.913 y=-525.366 z=464.12 mm, rx=-2.2348 ry=-2.2055 rz=-0.1004 rad; joints [-251.676, -74.86, 75.667, 270.873, -86.355, 109.144] deg
          Wait Sleep waitTime=1
          Call Check_Door_Open
          Switch expression=fail_flag
            Case (caseValue=0)
              Script: task_done = 1
            Case (caseValue=1)
              Script: retry_count = retry_count + 1
          Call Check_Camera_Open
          Switch expression=fail_flag
            Case (caseValue=0)
              Script: task_done = 1
            Case (caseValue=1)
              Script: retry_count = retry_count + 1
        If task_done == 0
          Call Error_Stop
        Wait Sleep waitTime=1
      Folder Task6,7:PickAndPlace
        Call Enter_Next_Task
        Loop While (checkContinuously=false) expression=retry_count <= max_retry and task_done == 0
          Folder Task6:PickA4FromScanner
            Call Enter_Next_Task
            MoveJ speed 60 deg/s, acceleration 80 deg/s^2 (useActiveTCP=true) feature=Base
              Waypoint Task6_Home: TCP in base x=258.69 y=-366.228 z=439.886 mm, rx=2.1238 ry=0.0367 rz=0.0867 rad; joints [-249.202, -96.956, 123.494, 186.236, -103.265, 192.053] deg
            MoveL speed 250 mm/s, acceleration 1200 mm/s^2 (useActiveTCP=true) feature=Base
              Waypoint Task6_Access: TCP in base x=313.846 y=-631.219 z=410.677 mm, rx=2.125 ry=0.0364 rz=0.0869 rad; joints [-253.141, -61.875, 85.575, 188.676, -99.891, 189.898] deg
            MoveL speed 250 mm/s, acceleration 1200 mm/s^2 (useActiveTCP=true) feature=Base
              Waypoint Pick2_1: TCP in base x=313.897 y=-687.473 z=339.098 mm, rx=2.1251 ry=0.0365 rz=0.0869 rad; joints [-254.541, -51.35, 79.738, 183.858, -98.731, 189.138] deg
              Waypoint Pick2_2: TCP in base x=297.062 y=-576.69 z=339.022 mm, rx=2.1252 ry=0.0365 rz=0.0869 rad; joints [-253.174, -63.627, 100.503, 175.507, -99.954, 189.881] deg
              Waypoint 웨이포인트_9: TCP in base x=297.068 y=-576.686 z=353.497 mm, rx=2.1253 ry=0.0365 rz=0.0869 rad; joints [-253.174, -64.796, 99.735, 177.449, -99.939, 189.883] deg
              Waypoint Pick2_3: TCP in base x=309.975 y=-404.431 z=313.224 mm, rx=1.5666 ry=0.061 rz=0.0686 rad; joints [-243.548, -63.004, 119.609, 123.351, -112.074, 180.495] deg
              Waypoint 웨이포인트_30: TCP in base x=304.477 y=-342.985 z=313.207 mm, rx=1.5667 ry=0.061 rz=0.0686 rad; joints [-239.92, -67.08, 127.258, 119.786, -115.719, 180.47] deg
              Waypoint 웨이포인트_31: TCP in base x=304.503 y=-342.949 z=162.635 mm, rx=1.5666 ry=0.0611 rz=0.0687 rad; joints [-239.873, -42.901, 125.648, 97.142, -115.787, 180.301] deg
              Waypoint 웨이포인트_32: TCP in base x=314.961 y=-460.117 z=158.017 mm, rx=1.5667 ry=0.0611 rz=0.0686 rad; joints [-246.074, -39.004, 110.38, 108.54, -109.568, 180.396] deg
              Waypoint 웨이포인트_33: TCP in base x=316.412 y=-476.469 z=181.081 mm, rx=1.5666 ry=0.061 rz=0.0686 rad; joints [-246.726, -41.395, 108.796, 112.519, -108.912, 180.428] deg
            Wait Sleep waitTime=1
            Call Gripper_Close
            Call Wait_Motor_Idle
            MoveL speed 250 mm/s, acceleration 1200 mm/s^2 (useActiveTCP=true) feature=Base
              Waypoint Task6_Retreat: TCP in base x=309.999 y=-343.473 z=344.222 mm, rx=1.5668 ry=0.0612 rz=0.0686 rad; joints [-239.216, -71.04, 125.629, 125.401, -116.4, 180.504] deg
            If fail_flag == 1
              Call Error_Stop
            Wait Sleep waitTime=1
          Folder Task7:PlaceA4InBasket
            MoveJ speed 60 deg/s, acceleration 80 deg/s^2 (useActiveTCP=true) feature=Base
              Waypoint Task7_Home: TCP in base x=310.006 y=-343.483 z=344.21 mm, rx=1.5668 ry=0.0612 rz=0.0685 rad; joints [-239.216, -71.037, 125.628, 125.4, -116.4, 180.503] deg
            MoveL speed 250 mm/s, acceleration 1200 mm/s^2 (useActiveTCP=true) feature=Base
              Waypoint Pick2_4: TCP in base x=310.007 y=-393.333 z=344.221 mm, rx=1.2229 ry=1.1845 rz=1.1938 rad; joints [-259.298, -65.163, 115.815, 127.425, -12.605, 182.2] deg
            MoveL speed 250 mm/s, acceleration 1200 mm/s^2 (useActiveTCP=true) feature=Base
              Waypoint 웨이포인트_18: TCP in base x=382.216 y=-393.345 z=344.199 mm, rx=1.2229 ry=1.1845 rz=1.1938 rad; joints [-250.278, -61.463, 109.361, 130.963, -21.61, 181.435] deg
              Waypoint 웨이포인트_22: TCP in base x=382.216 y=-393.346 z=344.196 mm, rx=1.5812 ry=1.549 rz=0.9034 rad; joints [-248.886, -78.626, 117.143, 195.783, -36.228, 131.246] deg
              Waypoint 웨이포인트_19: TCP in base x=454.461 y=-393.37 z=199.469 mm, rx=1.5812 ry=1.549 rz=0.9034 rad; joints [-241.291, -55.598, 113.717, 168.886, -41.185, 140.622] deg
              Waypoint 웨이포인트_10: TCP in base x=563.376 y=-393.348 z=166.569 mm, rx=1.6513 ry=1.6208 rz=0.8323 rad; joints [-231.558, -45.895, 98.537, 174.213, -51.411, 145.736] deg
              Waypoint 웨이포인트_11: TCP in base x=563.369 y=-393.371 z=166.52 mm, rx=1.8093 ry=1.7828 rz=0.6507 rad; joints [-230.388, -49.661, 98.443, 190.706, -60.696, 139.058] deg
            Call Gripper_Open
            Call Wait_Motor_Idle
            MoveL speed 250 mm/s, acceleration 1200 mm/s^2 (useActiveTCP=true) feature=Base
              Waypoint 웨이포인트_20: TCP in base x=549.465 y=-393.373 z=236.974 mm, rx=1.8092 ry=1.7828 rz=0.6507 rad; joints [-231.396, -57.67, 98.978, 198.671, -60.14, 138.047] deg
              Waypoint Task7_Retreat: TCP in base x=206.096 y=-224.681 z=522.613 mm, rx=0.5214 ry=0.8091 rz=-0.9024 rad; joints [-258.887, -102.991, 132.154, 112.549, -75.963, 106.161] deg
            Wait Sleep waitTime=1
            Call Check_Camera_Align
            Switch expression=paper_state
              Case (caseValue=0)
                Script: task_done = 1
              Case (caseValue=1)
                Script: retry_count = retry_count + 1
            Wait Sleep waitTime=1
        If task_done == 0
          Call Error_Stop
      Folder Task4:ClosePrinter
        Call Enter_Next_Task
        Loop While (checkContinuously=false) expression=retry_count <= max_retry and task_done == 0
          MoveJ speed 60 deg/s, acceleration 80 deg/s^2 (useActiveTCP=true) feature=Base
            Waypoint Task4_Home: TCP in base x=256.826 y=-439.474 z=610.895 mm, rx=2.3079 ry=0.0086 rz=0.0018 rad; joints [-252.464, -94.611, 91.606, 226.691, -102.422, 192.055] deg
          MoveL speed 250 mm/s, acceleration 1200 mm/s^2 (useActiveTCP=true) feature=Base
            Waypoint Task4_Access: TCP in base x=148.636 y=-727.715 z=605.166 mm, rx=1.2884 ry=-1.2507 rz=1.1591 rad; joints [-268.772, -57.066, 57.637, 184.345, -90.714, 269.314] deg
          MoveL speed 250 mm/s, acceleration 1200 mm/s^2 (useActiveTCP=true) feature=Base
            Waypoint Close1: TCP in base x=148.688 y=-809.891 z=547.115 mm, rx=1.4249 ry=-1.385 rz=1.0616 rad; joints [-268.907, -45.466, 43.512, 197.581, -90.443, 269.491] deg
            Waypoint Close2: TCP in base x=148.64 y=-796.037 z=521.65 mm, rx=1.4248 ry=-1.385 rz=1.0616 rad; joints [-268.893, -47.909, 51.494, 192.04, -90.504, 269.502] deg
            Waypoint Close3: TCP in base x=148.649 y=-796.055 z=521.571 mm, rx=1.6083 ry=-1.5658 rz=0.9063 rad; joints [-268.903, -50.476, 50.97, 209.943, -90.274, 269.718] deg
            Waypoint Close4: TCP in base x=148.687 y=-774.487 z=496.375 mm, rx=1.6083 ry=-1.5657 rz=0.9065 rad; joints [-268.873, -53.722, 60.073, 204.08, -90.336, 269.753] deg
            Waypoint Close5: TCP in base x=213.156 y=-749.245 z=470.417 mm, rx=1.6082 ry=-1.5657 rz=0.9065 rad; joints [-263.371, -54.366, 64.948, 200.023, -95.109, 272.561] deg
            Waypoint Close6: TCP in base x=213.168 y=-729.713 z=455.466 mm, rx=1.5446 ry=-1.5029 rz=0.9638 rad; joints [-263.137, -55.596, 71.043, 189.957, -95.666, 272.141] deg
            Waypoint 웨이포인트_2: TCP in base x=213.168 y=-700.447 z=569.635 mm, rx=1.5446 ry=-1.5029 rz=0.9637 rad; joints [-262.813, -62.268, 64.571, 203.117, -95.876, 272.261] deg
            Waypoint 웨이포인트_3: TCP in base x=213.139 y=-700.438 z=569.664 mm, rx=0.7687 ry=-0.7398 rz=1.4198 rad; joints [-262.888, -44.099, 47.902, 141.673, -95.592, 265.105] deg
            Waypoint 웨이포인트_4: TCP in base x=213.129 y=-710.201 z=438.633 mm, rx=0.7687 ry=-0.7398 rz=1.4198 rad; joints [-262.988, -38.166, 56.593, 127.044, -95.578, 265.084] deg
            Waypoint 웨이포인트_14: TCP in base x=213.137 y=-710.216 z=418.872 mm, rx=0.9791 ry=-0.9464 rz=1.3335 rad; joints [-262.867, -42.891, 66.704, 137.401, -96.512, 266.805] deg
            Waypoint 웨이포인트_15: TCP in base x=213.142 y=-710.217 z=394.52 mm, rx=1.1095 ry=-1.0745 rz=1.2674 rad; joints [-262.827, -44.827, 72.245, 143.715, -96.823, 268.018] deg
            Waypoint 웨이포인트_16: TCP in base x=213.146 y=-710.207 z=363.102 mm, rx=1.1858 ry=-1.1496 rz=1.2239 rad; joints [-262.817, -44.652, 75.673, 145.981, -96.899, 268.757] deg
          MoveL speed 250 mm/s, acceleration 1200 mm/s^2 (useActiveTCP=true) feature=Base
            Waypoint Task4_Retreat: TCP in base x=203.304 y=-382.609 z=703.619 mm, rx=0.9532 ry=-1.0966 rz=1.2827 rad; joints [-255.678, -95.084, 95.274, 165.571, -108.944, 268.685] deg
          Wait Sleep waitTime=1
          Call Check_Door_Closed
          Switch expression=fail_flag
            Case (caseValue=0)
              Script: task_done = 1
            Case (caseValue=1)
              Script: retry_count = retry_count + 1
        If task_done == 0
          Call Error_Stop
        Wait Sleep waitTime=1
    Folder Re_Init
      Call Init_Variables
      Script: global repeat = repeat + 1
      MoveJ speed 60 deg/s, acceleration 80 deg/s^2 (useActiveTCP=true) feature=Base
        Waypoint Home: TCP in base x=290.307 y=-472.673 z=405.346 mm, rx=-2.2604 ry=-2.147 rz=0.0783 rad; joints [-251.839, -82.418, 93.917, 258.527, -92.811, 111.318] deg
      Wait Sleep waitTime=1
SubProgram -> Socket_Open
SubProgram -> Init_Variables
SubProgram -> Gripper_Close
SubProgram -> Gripper_Open
SubProgram -> Wait_Motor_Idle
SubProgram -> Check_Door_Closed
SubProgram -> Check_Door_Open
SubProgram -> Check_Camera_Open
SubProgram -> Check_Camera_Align
SubProgram -> Error_Stop
SubProgram -> Enter_Next_Task
SubProgram Init_Variables (keepSynchronizedWithDisk=false)
  Script file /programs/usbdisk/새로운 폴더_3/Init_Variables.script
    | # ============================================================
    | # Init_Variables.script
    | # UR5e - PC Server - Arduino / PC Vision 공통 변수 초기화
    | # ============================================================
    | 
    | 
    | # ============================================================
    | # Retry / fail control
    | # ============================================================
    | 
    | global retry_count = 0
    | global max_retry = 2
    | 
    | global fail_flag = 0
    | global task_done = 0
    | global current_task = 0
    | 
    | global nopaper = 1
    | global align_retry_count = 0
    | 
    | # ============================================================
    | # State variables
    | # ============================================================
    | 
    | # Door sensor state
    | # 0: closed
    | # 1: open
    | global door_state = 0
    | 
    | # DC motor, Servo motor state
    | # 0: idle
    | # 1: busy
    | global motor_state = 0
    | 
    | # Scanner lid state
    | # 0: not open
    | # 1: open
    | global lid_state = 0
    | 
    | # Paper presence state
    | # 0: paper not found
    | # 1: paper present
    | global paper_state = 0
    | 
    | # Paper alignment state
    | # 0: OK
    | # 1: shifted up
    | # 2: shifted down
    | # 3: shifted left
    | # 4: shifted right
    | # 9: NG / unknown / not found
    | #
    | # 주의:
    | # PAPER_SHIFTED_*는 현재 종이가 벗어난 방향을 의미한다.
    | # 실제 보정 이동 방향은 반대다.
    | global paper_align_state = 9
    | 
    | 
    | # ============================================================
    | # Socket / response buffer
    | # ============================================================
    | 
    | global socket_state = False
    | global pc_response = ""
    | 
    | 
    | # ============================================================
    | # Command strings
    | # URScript -> PC Server -> Arduino / PC Vision
    | # ============================================================
    | 
    | # Arduino commands
    | global CMD_PING = "PING\n"
    | global CMD_GRIPPER_OPEN = "G OPEN\n"
    | global CMD_GRIPPER_CLOSE = "G CLOSE\n"
    | global CMD_DC_RUN = "D RUN\n"
    | global CMD_ESTOP = "ESTOP\n"
    | global CMD_MOTOR_STATUS = "MOTOR STATUS\n"
    | global CMD_DOOR_STATUS = "DOOR STATUS\n"
    | 
    | 
    | # PC Vision commands
    | global CMD_VISION_LID_STATUS = "V LID\n"
    | global CMD_VISION_PAPER_ALIGN = "V PAPER\n"
    | 
    | 
    | # ============================================================
    | # Expected Arduino response strings
    | # Arduino / PC Server -> URScript
    | # ============================================================
    | 
    | global RESP_OK_PING = "OK PING"
    | 
    | global RESP_OK_GRIPPER_OPEN = "OK G OPEN"
    | global RESP_OK_GRIPPER_CLOSE = "OK G CLOSE"
    | 
    | global RESP_OK_DC_RUN = "OK D RUN"
    | global RESP_OK_ESTOP = "OK ESTOP"
    | 
    | global RESP_MOTOR_BUSY = "MOTOR STATUS BUSY"
    | global RESP_MOTOR_IDLE = "MOTOR STATUS IDLE"
    | 
    | global RESP_DOOR_OPEN = "DOOR STATUS OPEN"
    | global RESP_DOOR_CLOSED = "DOOR STATUS CLOSED"
    | 
    | 
    | # ============================================================
    | # Expected PC Vision response strings: Lid
    | # PC Server -> URScript
    | # ============================================================
    | 
    | global RESP_LID_OPEN = "LID_OPEN"
    | global RESP_LID_CLOSED = "LID_CLOSED"
    | 
    | 
    | # ============================================================
    | # Expected PC Vision response strings: Paper alignment
    | # PC Server -> URScript
    | # ============================================================
    | 
    | global RESP_PAPER_OK = "PAPER_OK"
    | global RESP_PAPER_NOT_FOUND = "PAPER_NOT_FOUND"
    | 
    | global RESP_PAPER_SHIFTED_UP = "PAPER_SHIFTED_UP"
    | global RESP_PAPER_SHIFTED_DOWN = "PAPER_SHIFTED_DOWN"
    | global RESP_PAPER_SHIFTED_LEFT = "PAPER_SHIFTED_LEFT"
    | global RESP_PAPER_SHIFTED_RIGHT = "PAPER_SHIFTED_RIGHT"
    | global RESP_PAPER_NG = "PAPER_NG"
    | 
    | 
    | # ============================================================
    | # Optional common error response strings
    | # 현재는 unknown command 정도만 공통 확인용으로 둔다.
    | # Vision 내부 실패는 별도 ERR 없이 LID_CLOSED 또는 PAPER_NG로 처리한다.
    | # ============================================================
    | 
    | global RESP_ERR_UNKNOWN_CMD = "ERR UNKNOWN_CMD"
    | global RESP_ERR_ARDUINO_TIMEOUT = "ERR ARDUINO_TIMEOUT"
    | global RESP_ERR_ARDUINO_SERIAL = "ERR ARDUINO_SERIAL"
SubProgram Socket_Open (keepSynchronizedWithDisk=false)
  Script file /programs/usbdisk/새로운 폴더_2/Socket_Open.script
    | global socket_state = socket_open("192.168.0.10", 5000)
    | 
    | if socket_state:
    |   socket_send_string(CMD_PING)
    |   global pc_response = socket_read_line()
    | 
    |   if pc_response == RESP_OK_PING:
    |     global fail_flag = 0
    |     textmsg("Socket open OK")
    |   else:
    |     global fail_flag = 1
    |     textmsg("PING failed: ", pc_response)
    |   end
    | 
    | else:
    |   global fail_flag = 1
    |   textmsg("Socket open FAILED")
    |   halt
    | end
SubProgram Enter_Next_Task (keepSynchronizedWithDisk=false)
  Script file /programs/usbdisk/새로운 폴더_1/Enter_Next_Task.script
    | global current_task = current_task + 1
    | global retry_count = 0
    | global task_done = 0
    | global fail_flag = 0
SubProgram Check_Door_Open (keepSynchronizedWithDisk=false)
  Script file /home/ur/ursim-current/programs/0620_morning_UR5e_scripts/Check_Door_Open.script
    | socket_send_string(CMD_DOOR_STATUS)
    | global pc_response = socket_read_line()
    | 
    | if pc_response == RESP_DOOR_OPEN:
    |   global door_state = 1
    |   global fail_flag = 0
    | 
    | elif pc_response == RESP_DOOR_CLOSED:
    |   global door_state = 0
    |   global fail_flag = 1
    | 
    | else:
    |   global fail_flag = 1
    | end
SubProgram Check_Camera_Open (keepSynchronizedWithDisk=false)
  Script file /programs/usbdisk/새로운 폴더_3/Check_Camera_Open.script
    | # ============================================================
    | # Check_Camera_Open.script
    | # 목적:
    | # - PC Vision 서버에 V LID 명령 전송
    | # - ArUco 기반 스캐너 뚜껑 open/close 상태 확인
    | #
    | # 결과:
    | # - lid_state = 1 : LID_OPEN
    | # - lid_state = 0 : LID_CLOSED 또는 fail-safe
    | # - fail_flag = 0 : lid open 확인
    | # - fail_flag = 1 : lid open 아님
    | # ============================================================
    | 
    | socket_send_string(CMD_VISION_LID_STATUS)
    | global pc_response = socket_read_line()
    | 
    | if pc_response == RESP_LID_OPEN:
    |   global lid_state = 1
    |   global fail_flag = 0
    | 
    | elif pc_response == RESP_LID_CLOSED:
    |   global lid_state = 0
    |   global fail_flag = 1
    | 
    | else:
    |   global lid_state = 0
    |   global fail_flag = 1
    | end
SubProgram Error_Stop (keepSynchronizedWithDisk=false)
  Script file /home/ur/ursim-current/programs/0620_morning_UR5e_scripts/Error_Stop.script
    | # Arduino/PC 측 정지 요청을 먼저 수행
    | socket_send_string(CMD_ESTOP)
    | global pc_response = socket_read_line()
    | 
    | textmsg("ESTOP response: ", pc_response)
    | 
    | # 현재 task 번호에 따라 오류 메시지 출력
    | if current_task == 1:
    |   popup("Task 1 Failed: Open Printer", title="Task Error", warning=True, error=False)
    | 
    | elif current_task == 2:
    |   popup("Task 2 Failed: Pick A4 From Paper Box", title="Task Error", warning=True, error=False)
    | 
    | elif current_task == 3:
    |   popup("Task 3 Failed: Place A4 To Printer Head", title="Task Error", warning=True, error=False)
    | 
    | elif current_task == 4:
    |   popup("Task 4 Failed: Close Printer", title="Task Error", warning=True, error=False)
    | 
    | elif current_task == 5:
    |   popup("Task 5 Failed: Open Printer Again", title="Task Error", warning=True, error=False)
    | 
    | elif current_task == 6:
    |   popup("Task 6 Failed: Pick A4 From Printer Head", title="Task Error", warning=True, error=False)
    | 
    | elif current_task == 7:
    |   popup("Task 7 Failed: Place A4 To Paper Box", title="Task Error", warning=True, error=False)
    | 
    | elif current_task == 8:
    |   popup("Task 8 Failed: Close Printer Again", title="Task Error", warning=True, error=False)
    | 
    | else:
    |   popup("Unknown Task Failed", title="Task Error", warning=True, error=False)
    | end
    | 
    | halt # UR Program 정지
SubProgram Gripper_Open (keepSynchronizedWithDisk=false)
  Script file /programs/usbdisk/새로운 폴더_3/Gripper_Open.script
    | socket_send_string(CMD_GRIPPER_OPEN)
    | global pc_response = socket_read_line()
    | 
    | if pc_response == RESP_OK_GRIPPER_OPEN:
    |   global motor_state = 1
    |   global fail_flag = 0
    | 
    | else:
    |   global fail_flag = 1
    | end
SubProgram Wait_Motor_Idle (keepSynchronizedWithDisk=false)
  Script file /programs/usbdisk/새로운 폴더/Wait_Motor_Idle.script_bak
    | # MOTOR STATUS를 반복 조회하여 IDLE이 될 때까지 대기
    | # break문 사용 불가하므로 wait_done 임시 변수 사용
    | 
    | wait_done = 0
    | 
    | while wait_done == 0:
    |   socket_send_string(CMD_MOTOR_STATUS)
    |   global pc_response = socket_read_line()
    | 
    |   if pc_response == RESP_MOTOR_BUSY:
    |     global motor_state = 1
    |     sleep(0.1)
    | 
    |   elif pc_response == RESP_MOTOR_IDLE:
    |     global motor_state = 0
    |     global fail_flag = 0
    |     global wait_done = 1
    | 
    |   else:
    |     global fail_flag = 1
    |     global wait_done = 1
    |   end
    | end
SubProgram Gripper_Close (keepSynchronizedWithDisk=false)
  Script file /programs/usbdisk/새로운 폴더_3/Gripper_Close.script
    | socket_send_string(CMD_GRIPPER_CLOSE)
    | global pc_response = socket_read_line()
    | 
    | if pc_response == RESP_OK_GRIPPER_CLOSE:
    |   global motor_state = 1
    |   global fail_flag = 0
    | 
    | else:
    |   global fail_flag = 1
    | end
SubProgram Check_Camera_Align (keepSynchronizedWithDisk=false)
  Script file /programs/usbdisk/새로운 폴더_3/Check_Camera_Align.script
    | # ============================================================
    | # Check_Camera_Align.script
    | # 목적:
    | # - PC Vision 서버에 V PAPER 명령 전송
    | # - 종이 유무 및 정렬 상태 확인
    | #
    | # 결과:
    | # - paper_state = 1 : 종이 있음
    | # - paper_state = 0 : 종이 없음
    | #
    | # - paper_align_state = 0 : PAPER_OK
    | # - paper_align_state = 1 : PAPER_SHIFTED_UP
    | # - paper_align_state = 2 : PAPER_SHIFTED_DOWN
    | # - paper_align_state = 3 : PAPER_SHIFTED_LEFT
    | # - paper_align_state = 4 : PAPER_SHIFTED_RIGHT
    | # - paper_align_state = 9 : PAPER_NG / PAPER_NOT_FOUND / unknown
    | #
    | # 주의:
    | # - PAPER_SHIFTED_*는 현재 종이가 벗어난 방향이다.
    | # - 실제 보정 이동 방향은 반대다.
    | # ============================================================
    | 
    | socket_send_string(CMD_VISION_PAPER_ALIGN)
    | global pc_response = socket_read_line()
    | 
    | if pc_response == RESP_PAPER_OK:
    |   global paper_state = 1
    |   global paper_align_state = 0
    |   global fail_flag = 0
    | 
    | elif pc_response == RESP_PAPER_NOT_FOUND:
    |   global paper_state = 0
    |   global paper_align_state = 9
    |   global fail_flag = 1
    | 
    | elif pc_response == RESP_PAPER_SHIFTED_UP:
    |   global paper_state = 1
    |   global paper_align_state = 1
    |   global fail_flag = 1
    | 
    | elif pc_response == RESP_PAPER_SHIFTED_DOWN:
    |   global paper_state = 1
    |   global paper_align_state = 2
    |   global fail_flag = 1
    | 
    | elif pc_response == RESP_PAPER_SHIFTED_LEFT:
    |   global paper_state = 1
    |   global paper_align_state = 3
    |   global fail_flag = 1
    | 
    | elif pc_response == RESP_PAPER_SHIFTED_RIGHT:
    |   global paper_state = 1
    |   global paper_align_state = 4
    |   global fail_flag = 1
    | 
    | elif pc_response == RESP_PAPER_NG:
    |   global paper_state = 1
    |   global paper_align_state = 9
    |   global fail_flag = 1
    | 
    | else:
    |   global paper_state = 0
    |   global paper_align_state = 9
    |   global fail_flag = 1
    | end
SubProgram Check_Door_Closed (keepSynchronizedWithDisk=false)
  Script file /programs/usbdisk/새로운 폴더_3/Check_Door_Closed.script
    | socket_send_string(CMD_DOOR_STATUS)
    | global pc_response = socket_read_line()
    | 
    | if pc_response == RESP_DOOR_CLOSED:
    |   global door_state = 0
    |   global fail_flag = 0
    | 
    | elif pc_response == RESP_DOOR_OPEN:
    |   global door_state = 1
    |   global fail_flag = 1
    | 
    | else:
    |   global fail_flag = 1
    | end
